// TIA Portal V19 export
VAR_GLOBAL   // PLC tag table "U2Em4_Input"
   "null(34)" AT %I193.5 : Bool;   // 备用
   "null(27)" AT %I191.3 : Bool;   // 备用
   "null(40)" AT %I195.7 : Bool;   // 备用
   GripperCylinderHomePositionDetectionU2EM4_1 AT %I194.2 : Bool;   // U2EM4_ Clamping cylinder 1 in-situ detection / Em130_夹爪气缸1原位检测
   gripperCylinderWorkPositionDetectionOfSmallCellU2EM4_2 AT %I194.3 : Bool;   // U2EM4_clamp cylinder 2 small battery working position detection / Em130_夹爪气缸2小电池工作位检测
   withOrWithoutCellDetectionU2EM4_2 AT %I190.5 : Bool;   // U2EM4_Detect battery presence 2 / Em130_检测电池有无2
   GripperCylinderHomePositionDetectionU2EM4_3 AT %I195.0 : Bool;   // U2EM4_ Clamping cylinder 3 in-situ detection / Em130_夹爪气缸3原位检测
   yaxlEmotorOrgU2EM4 AT %I193.1 : Bool;   // U2EM4_Y-axis motor origin / Em130_Y轴电机原点
   yaxlEmotorPotU2EM4 AT %I192.7 : Bool;   // U2EM4_Y-axis motor positive limit / Em130_Y轴电机正限
   gripperCylinderWorkPositionDetectionOfSmallCellU2EM4_4 AT %I195.1 : Bool;   // U2EM4_clamp cylinder 4 small battery working position detection / Em130_夹爪气缸4小电池工作位检测
   handlingCollisionAvoidance2U2EM4 AT %I191.5 : Bool;   // U2EM4_Robot Collision Avoidance 2 / Em130_机械手防撞2
   gripperCylinderWorkPositionDetectionOfSmallCellU2EM4_3 AT %I194.6 : Bool;   // U2EM4_clamp cylinder 3 small battery working position detection / Em130_夹爪气缸3小电池工作位检测
   gripperCylinderWorkPositionDetectionOfBigCellU2EM4_3 AT %I194.7 : Bool;   // U2EM4_clamp cylinder 3 large battery working position detection / Em130_夹爪气缸3大电池工作位检测
   "null(42)" AT %I191.1 : Bool;   // 备用
   gripperCylinderWorkPositionDetectionOfBigCellU2EM4_2 AT %I194.4 : Bool;   // U2EM4_clamp cylinder 2 large battery working position detection / Em130_夹爪气缸2大电池工作位检测
   gripperCylinderWorkPositionDetectionOfBigCellU2EM4_1 AT %I194.1 : Bool;   // U2EM4_clamp cylinder 1 large battery working position detection / Em130_夹爪气缸1大电池工作位检测
   "null(39)" AT %I195.6 : Bool;   // 备用
   "null(33)" AT %I192.3 : Bool;   // 备用
   xaxlEmotorPotU2EM4 AT %I192.4 : Bool;   // U2EM4_X-axis motor positive limit / Em130_X轴电机正限
   zaxlEmotorNotU2EM4 AT %I193.3 : Bool;   // U2EM4_Z-axis motor negative limit / Em130_Z轴电机负限
   cellFoolproof4U2EM4 AT %I190.3 : Bool;   // U2EM4_Battery foolproof 4 / Em130_电池防呆4
   withOrWithoutCellDetectionU2EM4_3 AT %I190.6 : Bool;   // U2EM4_Detect battery presence 3 / Em130_检测电池有无3
   "null(30)" AT %I192.0 : Bool;   // 备用
   "null(35)" AT %I193.6 : Bool;   // 备用
   cellFoolproof1U2EM4 AT %I190.0 : Bool;   // U2EM4_Battery foolproof 1 / Em130_电池防呆1
   "null(41)" AT %I191.0 : Bool;   // 备用
   xaxlEmotorOrgU2EM4 AT %I192.6 : Bool;   // U2EM4_X-axis motor origin / Em130_X轴电机原点
   GripperCylinderHomePositionDetectionU2EM4_2 AT %I194.5 : Bool;   // U2EM4_ Clamping cylinder 2 in-situ detection / Em130_夹爪气缸2原位检测
   xaxlEmotorNotU2EM4 AT %I192.5 : Bool;   // U2EM4_X-axis motor negative limit / Em130_X轴电机负限
   handlingCollisionAvoidance4U2EM4 AT %I191.7 : Bool;   // U2EM4_Robot Collision Avoidance 4 / Em130_机械手防撞4
   handlingCollisionAvoidance3U2EM4 AT %I191.6 : Bool;   // U2EM4_Robot Collision Avoidance 3 / Em130_机械手防撞3
   zaxlEmotorPotU2EM4 AT %I193.2 : Bool;   // U2EM4_Z-axis motor positive limit / Em130_Z轴电机正限
   cellFoolproof3U2EM4 AT %I190.2 : Bool;   // U2EM4_Battery foolproof 3 / Em130_电池防呆3
   zaxlEmotorOrgU2EM4 AT %I193.4 : Bool;   // U2EM4_Z-axis motor origin / Em130_Z轴电机原点
   yaxlEmotorNotU2EM4 AT %I193.0 : Bool;   // U2EM4_Y-axis motor negative limit / Em130_Y轴电机负限
   handlingCollisionAvoidance1U2EM4 AT %I191.4 : Bool;   // U2EM4_Robot Collision Avoidance 1 / Em130_机械手防撞1
   cellFoolproof2U2EM4 AT %I190.1 : Bool;   // U2EM4_Battery foolproof 2 / Em130_电池防呆2
   gripperCylinderWorkPositionDetectionOfSmallCellU2EM4_1 AT %I194.0 : Bool;   // U2EM4_clamp cylinder 1 small battery working position detection / Em130_夹爪气缸1小电池工作位检测
   "null(31)" AT %I192.1 : Bool;   // 备用
   withOrWithoutCellDetectionU2EM4_4 AT %I190.7 : Bool;   // U2EM4_Detect battery presence 4 / Em130_检测电池有无4
   gripperCylinderWorkPositionDetectionOfBigCellU2EM4_4 AT %I195.2 : Bool;   // U2EM4_Clamping cylinder 4 large battery working position detection / Em130_夹爪气缸4大电池工作位检测
   GripperCylinderHomePositionDetectionU2EM4_4 AT %I195.3 : Bool;   // U2EM4_ Clamping cylinder 4 in-situ detection / Em130_夹爪气缸4原位检测
   withOrWithoutCellDetectionU2EM4_1 AT %I190.4 : Bool;   // U2EM4_Detect battery presence 1 / Em130_检测电池有无1
   "null(26)" AT %I191.2 : Bool;   // spare / 备用
   "null(36)" AT %I193.7 : Bool;   // spare / 备用
   "null(37)" AT %I195.4 : Bool;   // spare / 备用
   "null(32)" AT %I192.2 : Bool;   // spare / 备用
   "null(38)" AT %I195.5 : Bool;   // spare / 备用
END_VAR
